(* PLC project Blank Project, Blank Blank 1.0 *)
(* stored: creationDateTime 2016-05-18T21:14:07, modificationDateTime 2018-07-06T12:41:21 *)

PROGRAM My_Program
  VAR
    high_sensor_pin AT %IX0.3 : BOOL;
    flow_pin AT %QX0.0 : BOOL;
    low_sensor_pin AT %IX0.6 : BOOL;
    pump_pin AT %QX0.1 : BOOL;
  END_VAR

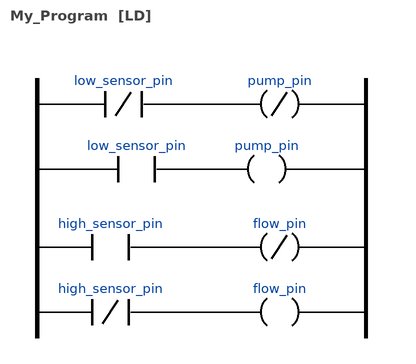
(* LD diagram, written out as Structured Text *)
pump_pin := NOT (NOT low_sensor_pin);
pump_pin := low_sensor_pin;
flow_pin := NOT high_sensor_pin;
flow_pin := NOT high_sensor_pin;
END_PROGRAM

CONFIGURATION Config0
  RESOURCE Res0 ON PLC
    TASK TaskMain(INTERVAL := T#5s0ms, PRIORITY := 0);
    PROGRAM Inst0 WITH TaskMain : My_Program;
  END_RESOURCE
END_CONFIGURATION
